Universal Robots PolyScope program: cb3_core_p1.urp

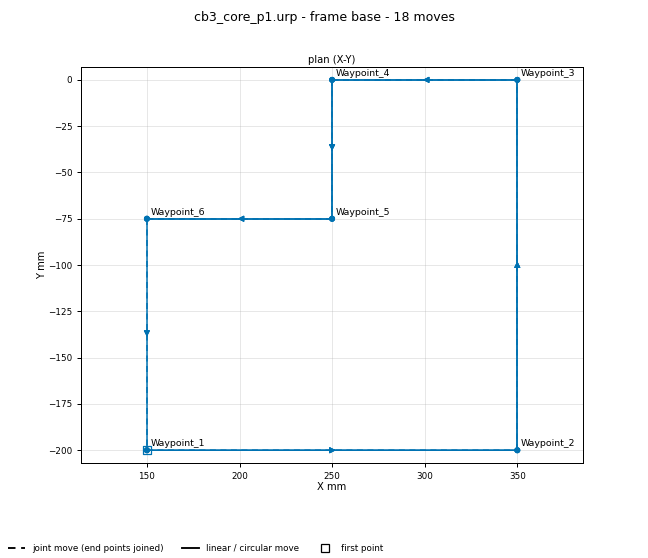
[picture p0: tool path of cb3_core_p1.urp in frame base, 18 of 18 moves have a stored position in this frame; points joined in program order, loops and branches not executed]
Program cb3_core_p1 (installation=default directory=/home/ur/ursim-current/programs createdIn=3.14.3.1031232 lastSavedIn=3.14.3.1031232 robotSerialNumber=2018339999)
Calibrated DH parameters: a=[0, -0.24365, -0.21325, 0, 0, 0]; d=[0.1519, 0, 0, 0.11235, 0.08535, 0.0819]; alpha=[1.570796, 0, 0, 1.570796, -1.570796, 0]; deltaTheta=[0, 0, 0, 0, 0, 0]
Robot Program (runOnlyOnce=false)
  MoveL speed 250 mm/s, acceleration 1200 mm/s^2 (useActiveTCP=true) feature=Base
    Waypoint Waypoint_1: TCP in base x=150 y=-199.999 z=100 mm, rx=0 ry=3.1416 rz=0 rad; joints [-26.425, -107.182, -144.788, -18.03, 90, 63.575] deg
    Waypoint Waypoint_2: TCP in base x=350 y=-199.995 z=100 mm, rx=0 ry=3.1416 rz=0 rad; joints [-13.561, -130.076, -97.112, -42.811, 90, 76.439] deg
    Waypoint Waypoint_3: motionParameters(blendRadius=0.05); TCP in base x=350 y=0 z=100 mm, rx=0 ry=3.1416 rz=0 rad; joints [18.723, -121.643, -114.663, -33.694, 90, 108.723] deg
    Waypoint Waypoint_4: motionParameters(blendRadius=0.025); TCP in base x=250 y=0 z=100 mm, rx=0 ry=3.1416 rz=0 rad; joints [26.705, -107.181, -144.787, -18.031, 90, 116.705] deg
    Waypoint Waypoint_5: motionParameters(blendRadius=0.025); TCP in base x=250 y=-75 z=100 mm, rx=0 ry=3.1416 rz=0 rad; joints [8.797, -108.737, -141.538, -19.725, 90, 98.797] deg
    Waypoint Waypoint_6: motionParameters(blendRadius=0.025); TCP in base x=150 y=-75 z=100 mm, rx=0 ry=3.1416 rz=0 rad; joints [15.496, -95.313, -170.223, -4.464, 90, 105.496] deg
  MoveJ speed 60 deg/s, acceleration 80 deg/s^2 (useActiveTCP=true)
    Waypoint Waypoint_1: TCP in base x=150 y=-199.999 z=100 mm, rx=0 ry=3.1416 rz=0 rad; joints [-26.425, -107.182, -144.788, -18.03, 90, 63.575] deg
    Waypoint Waypoint_2: TCP in base x=350 y=-199.995 z=100 mm, rx=0 ry=3.1416 rz=0 rad; joints [-13.561, -130.076, -97.112, -42.811, 90, 76.439] deg
    Waypoint Waypoint_3: TCP in base x=350 y=0 z=100 mm, rx=0 ry=3.1416 rz=0 rad; joints [18.723, -121.643, -114.663, -33.694, 90, 108.723] deg
    Waypoint Waypoint_4: TCP in base x=250 y=0 z=100 mm, rx=0 ry=3.1416 rz=0 rad; joints [26.705, -107.181, -144.787, -18.031, 90, 116.705] deg
    Waypoint Waypoint_5: TCP in base x=250 y=-75 z=100 mm, rx=0 ry=3.1416 rz=0 rad; joints [8.797, -108.737, -141.538, -19.725, 90, 98.797] deg
    Waypoint Waypoint_6: TCP in base x=150 y=-75 z=100 mm, rx=0 ry=3.1416 rz=0 rad; joints [15.496, -95.313, -170.223, -4.464, 90, 105.496] deg
  MoveP speed 250 mm/s, acceleration 1200 mm/s^2 (blendRadius=0.025 useActiveTCP=true) feature=Base
    Waypoint Waypoint_1: motionParameters(blendRadius=0.05); TCP in base x=150 y=-199.999 z=100 mm, rx=0 ry=3.1416 rz=0 rad; joints [-26.425, -107.182, -144.788, -18.03, 90, 63.575] deg
    Waypoint Waypoint_2: motionParameters(blendRadius=0.05); TCP in base x=350 y=-199.995 z=100 mm, rx=0 ry=3.1416 rz=0 rad; joints [-13.561, -130.076, -97.112, -42.811, 90, 76.439] deg
    Waypoint Waypoint_3: motionParameters(blendRadius=0.05); TCP in base x=350 y=0 z=100 mm, rx=0 ry=3.1416 rz=0 rad; joints [18.723, -121.643, -114.663, -33.694, 90, 108.723] deg
    Waypoint Waypoint_4: motionParameters(blendRadius=0.048); TCP in base x=250 y=0 z=100 mm, rx=0 ry=3.1416 rz=0 rad; joints [26.705, -107.181, -144.787, -18.031, 90, 116.705] deg
    Waypoint Waypoint_5: motionParameters(blendRadius=0.025); TCP in base x=250 y=-75 z=100 mm, rx=0 ry=3.1416 rz=0 rad; joints [8.797, -108.737, -141.538, -19.725, 90, 98.797] deg
    Waypoint Waypoint_6: motionParameters(blendRadius=0); TCP in base x=150 y=-75 z=100 mm, rx=0 ry=3.1416 rz=0 rad; joints [15.496, -95.313, -170.223, -4.464, 90, 105.496] deg
